(* PLC project Unnamed, Unknown Unnamed 1 *)
(* stored: creationDateTime 2026-05-01T21:20:24, modificationDateTime 2026-05-01T22:41:43 *)

PROGRAM proProject_03_Motor_Controlgram0
  VAR
    PB_EStop AT %IX0.0 : BOOL;
    PB_Stop AT %IX0.1 : BOOL;
    PB_Start AT %IX0.2 : BOOL;
    PB_FaultReset AT %IX0.3 : BOOL;
    SW_ModeAuto AT %IX0.4 : BOOL;
    F2_Overload AT %IX0.5 : BOOL;
    KM1_Feedback AT %IX0.6 : BOOL;
    KM_Star_Feedback AT %IX0.7 : BOOL;
    KM_Delta_Feedback AT %IX1.0 : BOOL;
    SEN_HighTemp AT %IX1.1 : BOOL;
    KM1_MainContactor AT %QX0.0 : BOOL;
    KM_Star AT %QX0.1 : BOOL;
    KM_Delta AT %QX0.2 : BOOL;
    HL1_RunLamp AT %QX0.3 : BOOL;
    HL2_StopLamp AT %QX0.4 : BOOL;
    HL3_AlarmLamp AT %QX0.5 : BOOL;
    HL4_StarLamp AT %QX0.6 : BOOL;
    HL5_DeltaLamp AT %QX0.7 : BOOL;
    MR_MasterEnable AT %MX0.0 : BOOL;
    MR_FaultOverload AT %MX0.1 : BOOL;
    MR_FaultHighTemp AT %MX0.2 : BOOL;
    MR_FaultContactor AT %MX0.3 : BOOL;
    MR_FaultAny AT %MX0.4 : BOOL;
    MR_RunLatch AT %MX0.5 : BOOL;
    MR_AutoMode AT %MX0.6 : BOOL;
    MR_ManualMode AT %MX0.7 : BOOL;
    MR_StarActive AT %MX1.0 : BOOL;
    MR_DeltaActive AT %MX1.1 : BOOL;
    MR_AutoStartCmd AT %MX1.2 : BOOL;
  END_VAR
  VAR
    StarDeltaTime : TIME := T#5s;
    FbkDelayTime : TIME := T#500s;
    TransDelayTime : TIME := T#200s;
    TON_FbkDelay : TON;
    TON_StarDelta : TON;
    TON_TransDelay : TON;
  END_VAR

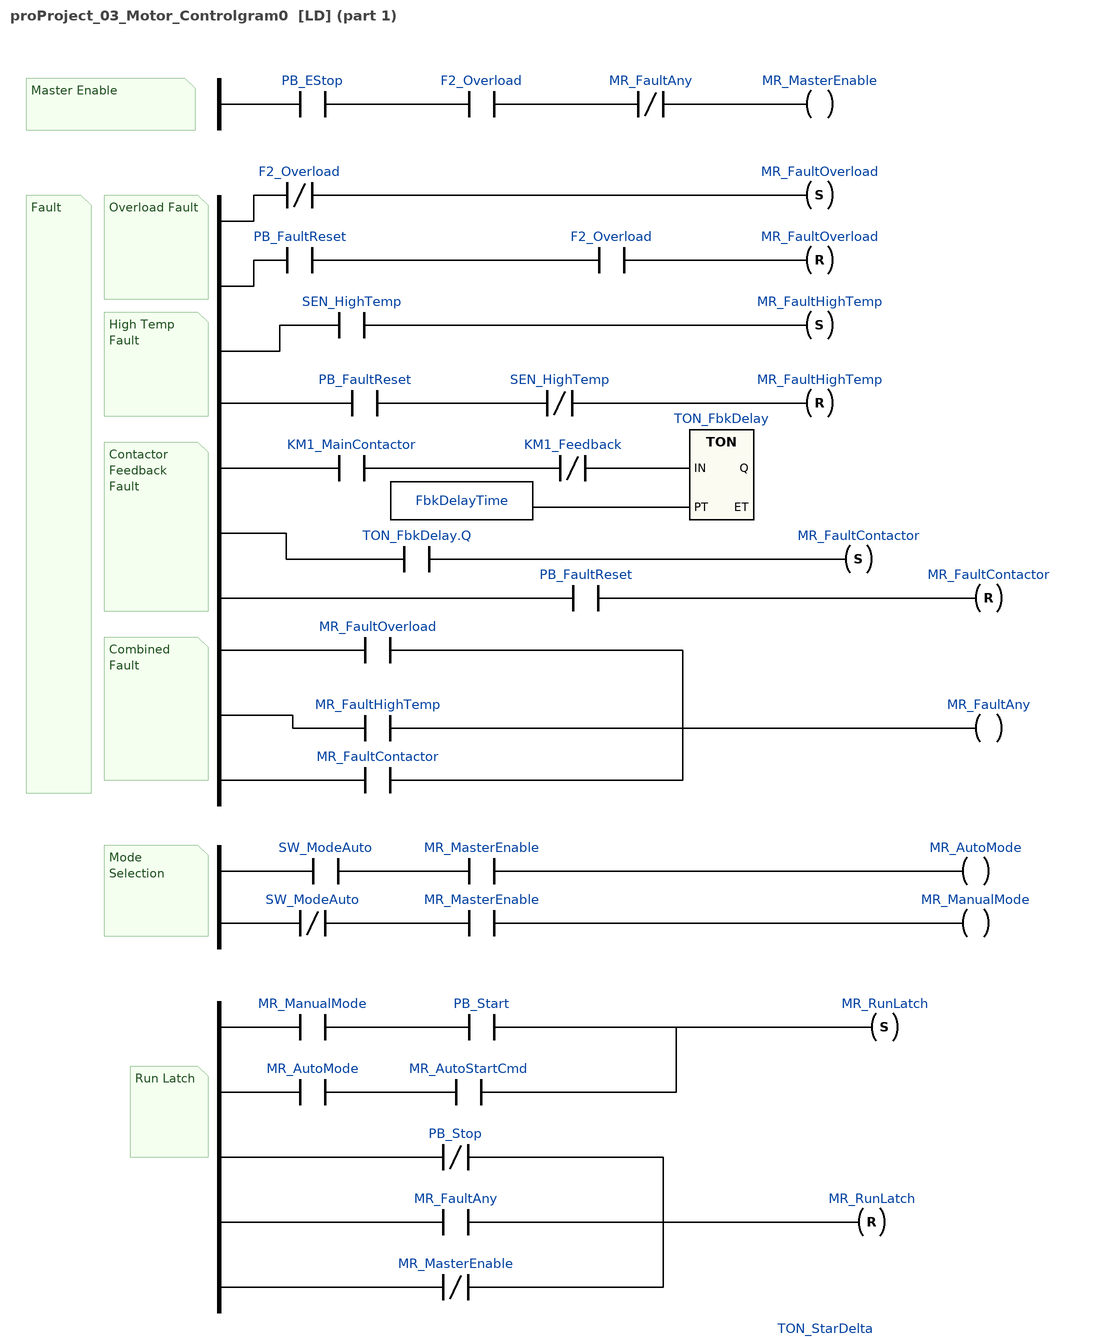
(* LD diagram, written out as Structured Text *)
(* Master Enable *)
MR_MasterEnable := PB_EStop AND F2_Overload AND NOT MR_FaultAny;
IF NOT F2_Overload THEN MR_FaultOverload := TRUE; END_IF;
(* Overload Fault *)
(* Fault *)
IF PB_FaultReset AND F2_Overload THEN MR_FaultOverload := FALSE; END_IF;
(* High Temp Fault *)
IF SEN_HighTemp THEN MR_FaultHighTemp := TRUE; END_IF;
IF PB_FaultReset AND NOT SEN_HighTemp THEN MR_FaultHighTemp := FALSE; END_IF;
(* Contactor Feedback Fault *)
IF TON_FbkDelay.Q THEN MR_FaultContactor := TRUE; END_IF;
IF PB_FaultReset THEN MR_FaultContactor := FALSE; END_IF;
(* Combined Fault *)
MR_FaultAny := MR_FaultHighTemp OR MR_FaultOverload OR MR_FaultContactor;
(* Mode Selection *)
MR_AutoMode := SW_ModeAuto AND MR_MasterEnable;
MR_ManualMode := NOT SW_ModeAuto AND MR_MasterEnable;
IF MR_ManualMode AND PB_Start OR MR_AutoMode AND MR_AutoStartCmd THEN MR_RunLatch := TRUE; END_IF;
(* Run Latch *)
IF MR_FaultAny OR NOT PB_Stop OR NOT MR_MasterEnable THEN MR_RunLatch := FALSE; END_IF;
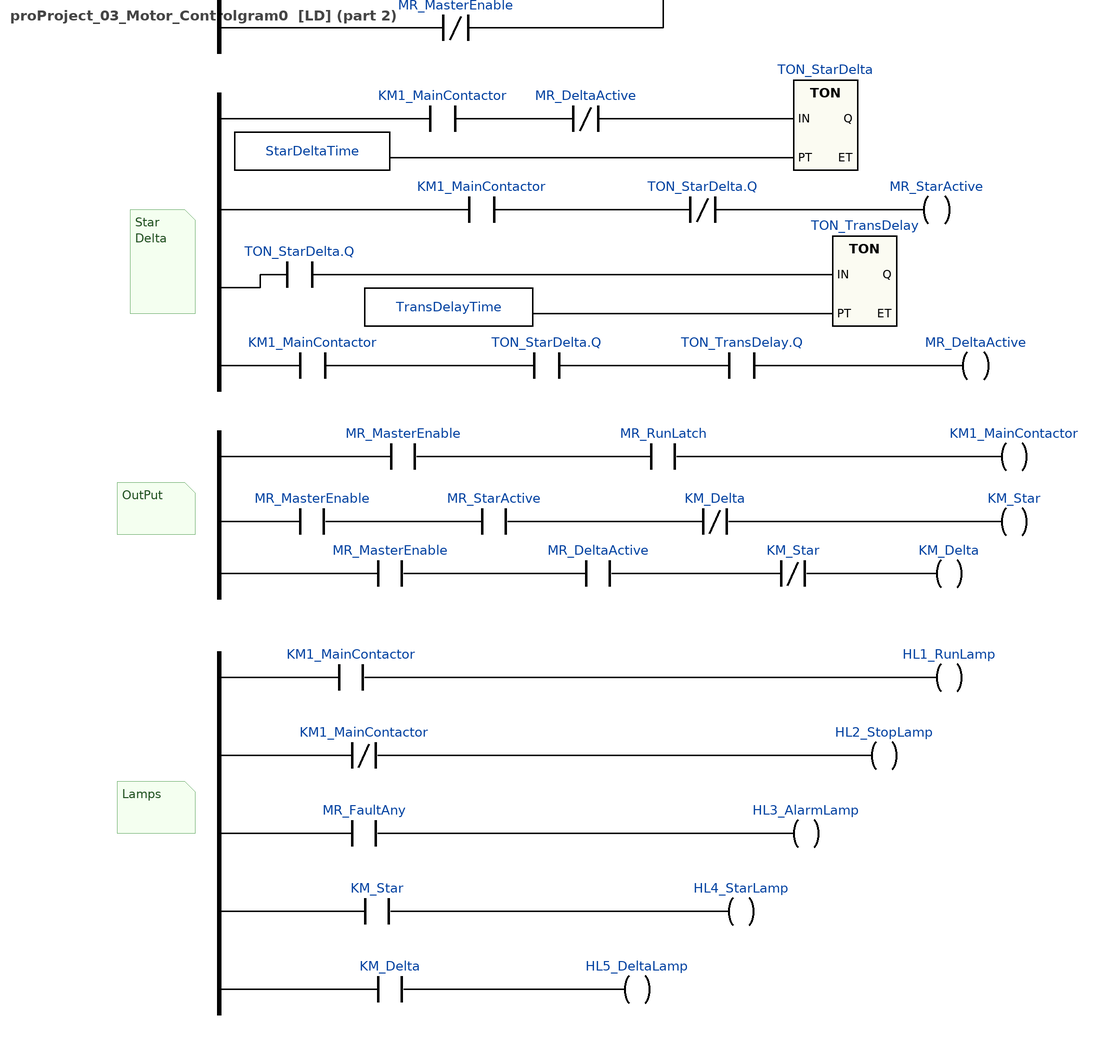
MR_StarActive := KM1_MainContactor AND NOT TON_StarDelta.Q;
(* Star Delta *)
MR_DeltaActive := KM1_MainContactor AND TON_StarDelta.Q AND TON_TransDelay.Q;
KM1_MainContactor := MR_MasterEnable AND MR_RunLatch;
(* OutPut *)
KM_Star := MR_MasterEnable AND MR_StarActive AND NOT KM_Delta;
KM_Delta := MR_MasterEnable AND MR_DeltaActive AND NOT KM_Star;
HL1_RunLamp := KM1_MainContactor;
HL2_StopLamp := NOT KM1_MainContactor;
(* Lamps *)
HL3_AlarmLamp := MR_FaultAny;
HL4_StarLamp := KM_Star;
HL5_DeltaLamp := KM_Delta;
TON_FbkDelay(IN := KM1_MainContactor AND NOT KM1_Feedback, PT := FbkDelayTime);
TON_StarDelta(IN := KM1_MainContactor AND NOT MR_DeltaActive, PT := StarDeltaTime);
TON_TransDelay(IN := TON_StarDelta.Q, PT := TransDelayTime);
END_PROGRAM

CONFIGURATION Config0
  RESOURCE Res0 ON PLC
    TASK task0(INTERVAL := T#20ms, PRIORITY := 0);
    PROGRAM instance0 WITH task0 : proProject_03_Motor_Controlgram0;
  END_RESOURCE
END_CONFIGURATION
